// TIA Portal V20 export
// export: Created 2025-12-01T14:57:23.8571024Z, ExportSetting None, DisplayName Totally Integrated Automation Portal, DisplayVersion V20 Update 3, DisplayName TIA Portal Openness, DisplayVersion V20 Update 3, DisplayName TIA Portal Version Control Interface, DisplayVersion V20 Update 3, DisplayName STEP 7 Professional, DisplayVersion V20 Update 3, DisplayName STEP 7 Safety, DisplayVersion V20 Update 2, DisplayName WinCC Basic/Comfort/Advanced, DisplayVersion V20 Update 3, DisplayName WinCC Professional, DisplayVersion V20 Update 3, DisplayName WinCC Unified, DisplayVersion V20 Update 3
DATA_BLOCK "DB013_ScadaZona"   // DB13
{ S7_Optimized_Access := 'FALSE' }
AUTHOR : SCADA
NAME : 20161001
VERSION : 1.0
// stored: AutoNumber false
   VAR
      Zona : Array[0.."CTE_MaxDispositivos"] of Struct
         Estado { S7_SetPoint := 'True'} : "EstadoZona";   // Estado de la Zona
         CodigoError : UDInt;
         Entradas { S7_SetPoint := 'True'} : "UDT_ScadaEntradasZona";
         Salidas { S7_SetPoint := 'True'} : "UDT_ScadaSalidasZona";
         DatosScada { S7_SetPoint := 'True'} : "UDT_ScadaDatosZona";
         EmergenciasGraves : Array[0..15] of Bool;
         EmergenciasLeves : Array[0..31] of Bool;
         ErroresGraves : Array[0..15] of Bool;
         ErroresLeves : Array[0..31] of Bool;
      END_STRUCT;
   END_VAR
BEGIN
END_DATA_BLOCK
